TYPE E_SAF_State :
(
	Control := 2,
	Run := 3
)UDINT;
END_TYPE

(* stored: Version 1.1.0.1, ProductVersion 3.1.4020.12
   DUT E_SAF_State: Id {f8b5ede6-3a93-4b2a-9e8e-d20feaac5ce7} *)
